FUNCTION_BLOCK E_MOVE (* Data latch (d) flip flop for ANY Datatype *)
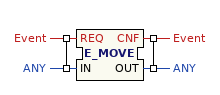
  EVENT_INPUT
    REQ WITH IN; (* Normal Execution Request *)
  END_EVENT
  EVENT_OUTPUT
    CNF WITH OUT; (* Execution Confirmation *)
  END_EVENT
  VAR_INPUT
    IN : ANY; (* input *)
  END_VAR
  VAR_OUTPUT
    OUT : ANY; (* input = output *)
  END_VAR
END_FUNCTION_BLOCK
